FUNCTION_BLOCK Piston
VAR_INPUT
	pSensor, nSensor : BOOL;
	pistonName : STRING;
END_VAR
VAR_OUTPUT
	pOut, nOut, error, isBusy : BOOL;
	errormessage: STRING(255);
	sState: STRING; // state of the piston
	isBKW: BOOL;
	isFWD: BOOL;
	isOFF: BOOL;
END_VAR
VAR
	_timeOut : TIME:= T#5S; // running the task timeout
	_delay : TIME:= T#1S; // in position (on sensor) timeout
	_noSensorTimeout : TIME:= T#2S; // sensor lost in FWD or BKW state
	timeOutTimer, delayTimer, noSensorTimeoutTimer : ton;
	state,task : ePiston;
	execute: BOOL; // run method with task input
	trExecute: R_trig;
	// testing rise error
	testError: BOOL; 
	//STEP mode - no use in this FB
	nextStep: BOOL;
	stepMode: BOOL;
	stepPB: BOOL;
	trStepPB: R_trig;
	sTask: STRING;
END_VAR

delayTimer(IN:= state=ePiston.running AND 
				(((task=ePiston.bkw) AND nSensor) OR
				((task=ePiston.fwd) AND pSensor)),
 		   PT:=_delay);
////////////////////////////////////////////////////////////////
timeOutTimer(IN:= state=ePiston.running AND
				  (((task=ePiston.bkw) AND NOT nSensor) OR 
				  ((task=ePiston.fwd) AND NOT pSensor)),
			 PT:=_timeOut);
////////////////////////////////////////////////////////////////
noSensorTimeoutTimer(IN:= (state=ePiston.fwd AND NOT pSensor) OR 
						  (state=episton.bkw AND NOT nSensor),
			 		 PT:= _noSensorTimeout );
////////////////////////////////////////////////////////////////
CASE state OF
	ePiston.off: // wait for execute trigger
		M_off();
	ePiston.running:
		IF M_run() THEN
			execute := FALSE;
			M_SetState(task);
		END_IF
	ePiston.fwd: // wait for execute trigger
		M_fwd();
	ePiston.bkw: // wait for execute trigger
		M_bkw();
	ePiston.error: // wait for reset method (from outside)
		M_off();
END_CASE
///////////////////////////////////////////////////////////////////////
statesIndication();
///////////////////////////////////////////////////////////////////////
trExecute(clk:=execute);
IF trExecute.Q AND state<>ePiston.error AND state<>ePiston.running THEN
			M_SetState(ePiston.running);
END_IF
///////////////////////////////////////////////////////////////////////
IF pSensor AND nSensor THEN
	M_riseError('- 2 sensors in one time - not acceptable!');
END_IF
///////////////////////////////////////////////////////////////////////
IF NOT error AND testError THEN // testing
	M_riseError('- testing error');
END_IF
///////////////////////////////////////////////////////////////////////
// STEP MODE
stepMode := FALSE; // STEP MODE not used
trStepPB(CLK:=stepPB);
nextStep := NOT stepMode OR trStepPB.Q; // for the M_SetState method  
///////////////////////////////////////////////////////////////////////

METHOD PUBLIC bkw : BOOL
VAR_INPUT
END_VAR
IF NOT execute AND state<>ePiston.error AND state<>ePiston.running
	AND state<>ePiston.bkw
	 THEN
	task := ePiston.bkw;
	execute := TRUE;
END_IF
END_METHOD

METHOD PUBLIC fwd : BOOL
VAR_INPUT
END_VAR
IF NOT execute AND state<>ePiston.error AND state<>ePiston.running
	AND state<>ePiston.fwd
	 THEN
	task := ePiston.fwd;
	execute := TRUE;
END_IF
END_METHOD

METHOD PRIVATE M_bkw : BOOL
VAR_INPUT
END_VAR
VAR
	//bkwState : BOOL;
END_VAR
pout := FALSE;
nout := TRUE;

IF state=ePiston.bkw AND (noSensorTimeoutTimer.Q OR pSensor) THEN
	M_riseError('- error in BKW - check the sensor');
END_IF
END_METHOD

METHOD PRIVATE M_fwd : BOOL
VAR_INPUT
END_VAR
VAR
	//fwdState : BOOL;
END_VAR
pout := TRUE;
nout := FALSE;

IF state=ePiston.fwd AND (noSensorTimeoutTimer.Q OR nSensor) THEN
	M_riseError('- error in FWD - check the sensor');
END_IF
END_METHOD

METHOD PRIVATE M_off : BOOL
VAR_INPUT
END_VAR
pOut := FALSE;
nOut := FALSE;
END_METHOD

METHOD PRIVATE M_riseError : BOOL
VAR_INPUT
	message : STRING;
END_VAR
errormessage := CONCAT(pistonName, message);

IF NOT error THEN
	error := TRUE;
	M_SetState(episton.error);
	//TODO log with message
END_IF
END_METHOD

METHOD PRIVATE M_run : BOOL
VAR_INPUT
	//task : INT; // enum
END_VAR
CASE task OF
	ePiston.off:
		M_off();
		M_run := TRUE;
	ePiston.bkw:
		M_bkw();
	ePiston.fwd:
		M_fwd();
END_CASE
sTask := stateToString(task);

IF delayTimer.Q THEN
	sTask := '';
	M_run := TRUE;
ELSIF timeOutTimer.Q THEN
	M_riseError(CONCAT('- timeout in the task: ' , stateToString(task)));
END_IF
END_METHOD

METHOD PRIVATE M_SetState
VAR_INPUT
	eNextState : ePiston; //INT;
END_VAR
IF State <> eNextState AND nextStep THEN
	//AddEventToLog(State,SeverityLevelType.Info,f_concat9( 'Changing State FROM ', M_statetostring(State), 'TO' ,M_StateToString(eNextState),'','','','',''));
	State := eNextState;
	//stateString := M_statetostring(State);
END_IF
END_METHOD

METHOD PUBLIC off : BOOL
VAR_INPUT
END_VAR
IF NOT execute AND state<>ePiston.error AND state<>ePiston.running 
	AND state<>ePiston.off
	THEN
	task := ePiston.off;
	execute := TRUE;
END_IF
END_METHOD

METHOD reset : BOOL
VAR_INPUT
END_VAR
IF state = episton.error OR error THEN
	M_SetState(ePiston.off);
	execute := FALSE;
	error := FALSE;
	errormessage := '';
END_IF
END_METHOD

METHOD PUBLIC setTimers : BOOL
VAR_INPUT
	timeOut : TIME; // running the task timeout
	delay : TIME; // in position (on sensor) timeout
	noSensorTimeout : TIME; // sensor lost in FWD or BKW state
END_VAR
_timeOut			:= timeOut;
_delay				:= delay;
_noSensorTimeout	:= noSensorTimeout;
END_METHOD

ACTION statesIndication:
isBKW := state = ePiston.bkw;
isFWD := state = ePiston.fwd;
isOFF := state = ePiston.off;
isBusy := state = ePiston.running;

sState := stateToString(state);
END_ACTION

METHOD PRIVATE stateToString : string
VAR_INPUT
	ePistonState : INT; // ePiston enum
END_VAR
CASE ePistonState OF
	ePiston.bkw:
		stateToString := 'BKW';
	ePiston.fwd:
		stateToString := 'FWD';
	ePiston.error:
		stateToString := 'ERROR';
	ePiston.off:
		stateToString := 'OFF';
	ePiston.running:
		stateToString :=concat('RUNNING ', sTask);
END_CASE
END_METHOD

END_FUNCTION_BLOCK

(* stored: Version 1.1.0.1, ProductVersion 3.1.4022.18
   POU Piston: Id {c14a18be-a5d9-43d9-b57d-de6b138fcbb5}, SpecialFunc None
   Folder PRIVATE: Id {61449881-cae0-4ebb-b34b-72e2db08101a}
   Folder PUBLIC: Id {4020de6b-bfe2-4690-90ea-5b2ee17be787}
   Method bkw: Id {824a11d5-4a48-469b-931c-511dd1b840fd}
   Method fwd: Id {0a956e4d-e0bc-4c11-a9b7-662ed6e9c9a2}
   Method M_bkw: Id {3af92d9f-7b09-4f80-84a4-104ebc223884}
   Method M_fwd: Id {54d50cd5-59ac-4917-90e2-80082ce6663f}
   Method M_off: Id {bdccd2e6-762d-498f-b2f6-acc0769d10ce}
   Method M_riseError: Id {7a55061b-e795-4356-8e11-89a70f30e0ac}
   Method M_run: Id {1d65d539-57ff-42ab-905f-08e897f1c7ef}
   Method M_SetState: Id {fff2b4ea-d767-4297-83f8-a3b94f560f77}
   Method off: Id {78b1207f-ec0c-4c4c-87dd-ed6889887f33}
   Method reset: Id {f4efaf27-7af3-4aa9-a520-b46aadb0ac18}
   Method setTimers: Id {4bdac6d6-8ff1-4608-9e37-15cf81dc8ae2}
   Action statesIndication: Id {f499436d-ad82-4e21-a113-f5972912f63c}
   Method stateToString: Id {66c0262a-ead9-42bb-aedb-1a3dcb5e8ca8} *)
